FUNCTION_BLOCK FB_ADSWatchdog
VAR
    _tZoneA     : TON;
    _tZoneB     : TON;
    _tZoneC     : TON;
    _bZoneAOk   : BOOL := FALSE;
    _bZoneBOk   : BOOL := FALSE;
    _bZoneCOk   : BOOL := FALSE;
END_VAR
VAR_INPUT
    bZoneACommOk : BOOL;    // from FB_ADSZoneReader Zone A
    bZoneBCommOk : BOOL;    // from FB_ADSZoneReader Zone B
    bZoneCCommOk : BOOL;    // from FB_ADSZoneReader Zone C
END_VAR
VAR_OUTPUT
    bZoneAHealthy   : BOOL;
    bZoneBHealthy   : BOOL;
    bZoneCHealthy   : BOOL;
    bAllZonesHealthy : BOOL;
    bAnyZoneLost    : BOOL;
END_VAR

// FB Body
// ─────────────────────────────────────
// Each zone gets independent watchdog
// Loss of comm held for debounce period
// before declaring zone lost
// ─────────────────────────────────────
_tZoneA(
    IN := NOT bZoneACommOk,
    PT := GVL_SafetyLimits.c_tADS_WATCHDOG
);

_tZoneB(
    IN := NOT bZoneBCommOk,
    PT := GVL_SafetyLimits.c_tADS_WATCHDOG
);

_tZoneC(
    IN := NOT bZoneCCommOk,
    PT := GVL_SafetyLimits.c_tADS_WATCHDOG
);

// Zone healthy if watchdog has NOT timed out
bZoneAHealthy    := NOT _tZoneA.Q;
bZoneBHealthy    := NOT _tZoneB.Q;
bZoneCHealthy    := NOT _tZoneC.Q;

bAllZonesHealthy := bZoneAHealthy
                AND bZoneBHealthy
                AND bZoneCHealthy;

bAnyZoneLost     := NOT bZoneAHealthy
                 OR NOT bZoneBHealthy
                 OR NOT bZoneCHealthy;

END_FUNCTION_BLOCK

(* stored: Version 1.1.0.1, ProductVersion 3.1.4024.16
   POU FB_ADSWatchdog: Id {9038667c-cc3b-4480-9285-5726ae5e9b38}, SpecialFunc None *)
